/// This struct contains variables that
/// * are read from outside (e.g. HMI) to retrieve information about the unit's current state and (temporary) parameters (= `publish`) 
/// * are written from outside (e.g. HMI) to control the unit via ADS (= `subscribe`) 
TYPE MachineCom :
STRUCT
  Publish : MachineComPublish;
  Subscribe : MachineComSubscribe;
END_STRUCT
END_TYPE

(* stored: Version 1.1.0.1
   DUT MachineCom: Id {bdb876af-bae3-41c3-9b6e-85370b234033} *)
